Staubli VAL3: setIO.pgx

public program setIO(string x_sIO)
begin
  //
  sIOName=x_sIO
end
